{attribute addProperty BoxType "EK1122-0000-0018"}
{attribute addProperty Id "Beckhoff_EQ3xxxsub_EK1100EK1100_179A0949162A_0001_EQ3174_0002_0016EQ3174_55F04E9922428A_0002_EQ3174_0002_0017EQ3174_55F04E9922428A_0003_EQ3174_0002_0021EQ3174_55F04E9922428A_0004_EQ3174_0002_0022EQ3174_83515A0D22428A_0005_EQ3174_0002_0023EQ3174_83515A0D22428A_0006_EQ3204_0002_0016EQ3204_BF093E1239249A_0007_EQ3204_0002_0017EQ3204_BF093E1239249A_0008_EQ3204_0002_0020EQ3204_BF093E1239249A_0009_EQ3204_0002_0021EQ3204_69AA4F8E22428A_0010_EQ3204_0002_0022EQ3204_69AA4F8E22428A_0011_EQ3314_0002_0016EQ3314_AF8E369F22428A_0012_EQ3314_0002_0017EQ3314_AF8E369F22428A_0013_EQ3314_0002_0021EQ3314_AF8E369F22428A_0014_EQ3314_0002_0022EQ3314_2E54E3B022428"}
{attribute addProperty CRC "871053013"}
{attribute addProperty SizeInBites "3656"}
{attribute addProperty SizeInBytes "457"}
TYPE Beckhoff_EQ3xxxEK1122_33EB36D5 EXTENDS EK1122_179A0949 :
STRUCT
	{attribute addProperty Name "Beckhoff_EQ3xxxsub_EK1100"}
	Beckhoff_EQ3xxxsub_EK1100 : EK1100_179A0949;
	{attribute addProperty Name "A_0001_EQ3174_0002_0016"}
	A_0001_EQ3174_0002_0016 : EQ3174_55F04E99;
	{attribute addProperty Name "A_0002_EQ3174_0002_0017"}
	A_0002_EQ3174_0002_0017 : EQ3174_55F04E99;
	{attribute addProperty Name "A_0003_EQ3174_0002_0021"}
	A_0003_EQ3174_0002_0021 : EQ3174_55F04E99;
	{attribute addProperty Name "A_0004_EQ3174_0002_0022"}
	A_0004_EQ3174_0002_0022 : EQ3174_83515A0D;
	{attribute addProperty Name "A_0005_EQ3174_0002_0023"}
	A_0005_EQ3174_0002_0023 : EQ3174_83515A0D;
	{attribute addProperty Name "A_0006_EQ3204_0002_0016"}
	A_0006_EQ3204_0002_0016 : EQ3204_BF093E12;
	{attribute addProperty Name "A_0007_EQ3204_0002_0017"}
	A_0007_EQ3204_0002_0017 : EQ3204_BF093E12;
	{attribute addProperty Name "A_0008_EQ3204_0002_0020"}
	A_0008_EQ3204_0002_0020 : EQ3204_BF093E12;
	{attribute addProperty Name "A_0009_EQ3204_0002_0021"}
	A_0009_EQ3204_0002_0021 : EQ3204_69AA4F8E;
	{attribute addProperty Name "A_0010_EQ3204_0002_0022"}
	A_0010_EQ3204_0002_0022 : EQ3204_69AA4F8E;
	{attribute addProperty Name "A_0011_EQ3314_0002_0016"}
	A_0011_EQ3314_0002_0016 : EQ3314_AF8E369F;
	{attribute addProperty Name "A_0012_EQ3314_0002_0017"}
	A_0012_EQ3314_0002_0017 : EQ3314_AF8E369F;
	{attribute addProperty Name "A_0013_EQ3314_0002_0021"}
	A_0013_EQ3314_0002_0021 : EQ3314_AF8E369F;
	{attribute addProperty Name "A_0014_EQ3314_0002_0022"}
	A_0014_EQ3314_0002_0022 : EQ3314_2E54E3B0;
END_STRUCT
END_TYPE

(* stored: Version 1.2.0.0, ProductVersion 3.1.4024.9
   DUT Beckhoff_EQ3xxxEK1122_33EB36D5: Id {900832e4-7ac1-42f5-ae31-293b187811e6} *)
